SUBAPPLICATION Verteiler (* Subapplication Type *)
  (* Standard: 61499-2 *)
  (* Version 1.0, 2023-01-29, Franz *)
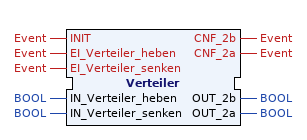
  EVENT_INPUT
    INIT;
    EI_Verteiler_heben;
    EI_Verteiler_senken;
  END_EVENT
  EVENT_OUTPUT
    CNF_2b;
    CNF_2a;
  END_EVENT
  VAR_INPUT
    IN_Verteiler_heben : BOOL;
    IN_Verteiler_senken : BOOL;
  END_VAR
  VAR_OUTPUT
    OUT_2b : BOOL;
    OUT_2a : BOOL;
  END_VAR
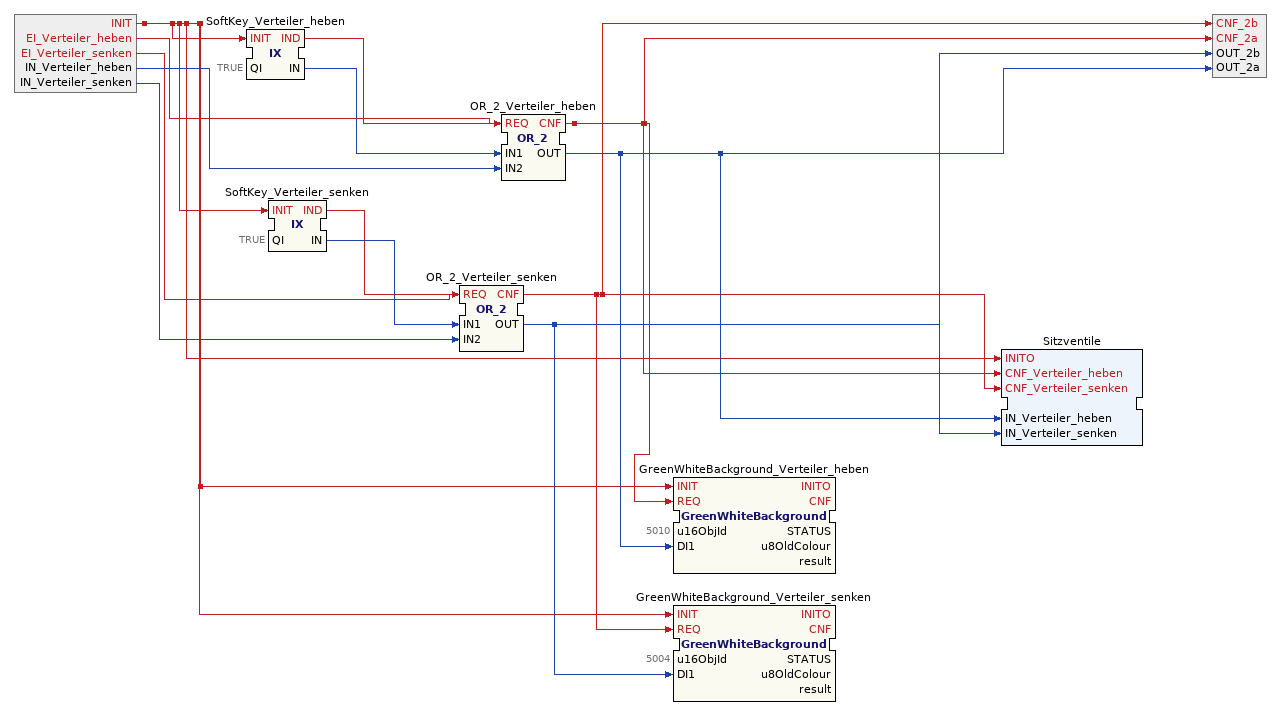
  FBS
    OR_2_Verteiler_senken : OR_2;
    SoftKey_Verteiler_heben : IX(QI := TRUE);
    OR_2_Verteiler_heben : OR_2;
    GreenWhiteBackground_Verteiler_heben : GreenWhiteBackground(u16ObjId := 5010);
    SoftKey_Verteiler_senken : IX(QI := TRUE);
    GreenWhiteBackground_Verteiler_senken : GreenWhiteBackground(u16ObjId := 5004);
  END_FBS
  SUBAPPLICATION Sitzventile (* Sitzventile *)
    EVENT_INPUT
      INITO;
      CNF_Verteiler_heben;
      CNF_Verteiler_senken;
    END_EVENT
    VAR_INPUT
      IN_Verteiler_heben : BOOL;
      IN_Verteiler_senken : BOOL;
    END_VAR
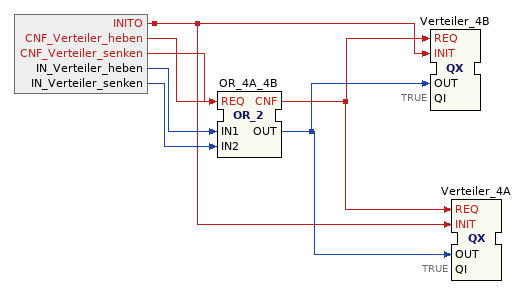
    FBS
      OR_4A_4B : OR_2; {SET_ATTRIBUTE(PinComment, IN1:Verteiler_heben)} {SET_ATTRIBUTE(PinComment, IN2:Verteiler_senken)}
      Verteiler_4B : QX(QI := TRUE);
      Verteiler_4A : QX(QI := TRUE);
    END_FBS
    EVENT_CONNECTIONS
      OR_4A_4B.CNF TO Verteiler_4B.REQ;
      OR_4A_4B.CNF TO Verteiler_4A.REQ;
      CNF_Verteiler_heben TO OR_4A_4B.REQ;
      CNF_Verteiler_senken TO OR_4A_4B.REQ;
      INITO TO Verteiler_4B.INIT;
      INITO TO Verteiler_4A.INIT;
    END_CONNECTIONS
    DATA_CONNECTIONS
      OR_4A_4B.OUT TO Verteiler_4B.OUT;
      OR_4A_4B.OUT TO Verteiler_4A.OUT;
      IN_Verteiler_heben TO OR_4A_4B.IN1;
      IN_Verteiler_senken TO OR_4A_4B.IN2;
    END_CONNECTIONS
  END_SUBAPPLICATION
  EVENT_CONNECTIONS
    SoftKey_Verteiler_senken.IND TO OR_2_Verteiler_senken.REQ;
    SoftKey_Verteiler_heben.IND TO OR_2_Verteiler_heben.REQ;
    OR_2_Verteiler_heben.CNF TO GreenWhiteBackground_Verteiler_heben.REQ;
    INIT TO SoftKey_Verteiler_heben.INIT;
    INIT TO SoftKey_Verteiler_senken.INIT;
    INIT TO Sitzventile.INITO;
    OR_2_Verteiler_senken.CNF TO GreenWhiteBackground_Verteiler_senken.REQ;
    INIT TO GreenWhiteBackground_Verteiler_heben.INIT;
    INIT TO GreenWhiteBackground_Verteiler_senken.INIT;
    OR_2_Verteiler_heben.CNF TO Sitzventile.CNF_Verteiler_heben;
    OR_2_Verteiler_senken.CNF TO Sitzventile.CNF_Verteiler_senken;
    EI_Verteiler_heben TO OR_2_Verteiler_heben.REQ;
    EI_Verteiler_senken TO OR_2_Verteiler_senken.REQ;
    OR_2_Verteiler_heben.CNF TO CNF_2a;
    OR_2_Verteiler_senken.CNF TO CNF_2b;
  END_CONNECTIONS
  DATA_CONNECTIONS
    SoftKey_Verteiler_senken.IN TO OR_2_Verteiler_senken.IN1;
    SoftKey_Verteiler_heben.IN TO OR_2_Verteiler_heben.IN1;
    OR_2_Verteiler_heben.OUT TO GreenWhiteBackground_Verteiler_heben.DI1;
    IN_Verteiler_senken TO OR_2_Verteiler_senken.IN2;
    IN_Verteiler_heben TO OR_2_Verteiler_heben.IN2;
    OR_2_Verteiler_heben.OUT TO Sitzventile.IN_Verteiler_heben;
    OR_2_Verteiler_senken.OUT TO Sitzventile.IN_Verteiler_senken;
    OR_2_Verteiler_senken.OUT TO GreenWhiteBackground_Verteiler_senken.DI1;
    OR_2_Verteiler_heben.OUT TO OUT_2a;
    OR_2_Verteiler_senken.OUT TO OUT_2b;
  END_CONNECTIONS
END_SUBAPPLICATION
